TYPE DUT_Rexroth_Parameter :
STRUCT
	Beschleunigung	:LREAL;
	Verzoegerung	:LREAL;
	Ruck			:LREAL;
END_STRUCT
END_TYPE

(* stored: Version 1.1.0.1
   DUT DUT_Rexroth_Parameter: Id {c86ae7f1-f068-4264-a5de-7b48ac91967d} *)
